TYPE WrappedComponentExample_Control EXTENDS TcoCore.TcoStruct :
STRUCT
    Setpoint : INT;
END_STRUCT
END_TYPE

(* stored: Version 1.1.0.1, ProductVersion 3.1.4024.12
   DUT WrappedComponentExample_Control: Id {381cd645-ffa5-0c7b-2bf4-2303d6818f94} *)
